TYPE ST_MethodOut :  //    方法
STRUCT
             Execute            :BOOL;  
             Done1               :BOOL;  
             Done2               :BOOL;  
             Error               :BOOL;

END_STRUCT
END_TYPE

(* stored: Version 1.1.0.1, ProductVersion 3.1.4024.9
   DUT ST_MethodOut: Id {f541868b-93b9-4a2b-a408-12012db56f6b} *)
